// TIA Portal V17 export
// export: Created 2026-08-06T00:00:00, ExportSetting ResearchOS test fixture
BLOCK "FB_Motor"   // ObjectSW100, LAD
// Motor control with self-holding circuit
BEGIN

REGION Network 1: Self-holding motor start
END_REGION
END_BLOCK
